// TIA Portal V16 export
// export: Created 2024-12-03T15:41:41.0204525Z, ExportSetting WithDefaults, DisplayName Totally Integrated Automation Portal, DisplayVersion V16 Update 6, DisplayName TIA Portal Version Control Interface, DisplayVersion V16 Update 2, DisplayName TIA Portal Openness, DisplayVersion V16 Update 6, DisplayName TIA Portal Teamcenter Gateway, DisplayVersion V16, DisplayName SINAMICS Startdrive Advanced, DisplayVersion V16 Update 5, DisplayName SINAMICS Startdrive G130, G150, S120, S150, SINAMICS MV, S210, DisplayVersion V16 Update 5, DisplayName SINAMICS Startdrive G110M, G120, G120C, G120D, G120P, G115D, DisplayVersion V16 Update 5, DisplayName STEP 7 Professional, DisplayVersion V16 Update 6, DisplayName STEP 7 Safety, DisplayVersion V16, DisplayName WinCC Advanced / Unified PC, DisplayVersion V16 Update 6
FUNCTION_BLOCK "ScanTimer_FB"   // FB42, SCL
{ S7_Optimized_Access := 'TRUE' }
VERSION : 0.1
// stored: AutoNumber true, IsIECCheckEnabled false, IsRetainMemResEnabled false, MemoryReserve 100, SetENOAutomatically false, UDAEnableTagReadback false
   VAR_OUTPUT
      O_ScanTime : DInt;
   END_VAR
   VAR
      PrevDate : DInt;
   END_VAR
   VAR_TEMP
      T_Date : DTL;
      T_Res : Int;
      T_CurrentDate : DInt;
      T_diff : DInt;
   END_VAR
BEGIN
   REGION _name_

       #T_Res := RD_SYS_T(#T_Date);
       #T_CurrentDate := TOD_TO_DINT(DTL_TO_TOD(#T_Date));
       #T_diff := #T_CurrentDate - #PrevDate;

       IF (#T_diff > 0) THEN
           #O_ScanTime := #T_diff;
       END_IF;

       #PrevDate := #T_CurrentDate;

   END_REGION
END_FUNCTION_BLOCK
